# EPICS substitutions: plotApp/Db/plot.substitutions
# P comes from epicsEnvSet("P", ...) in st.cmd (e.g. TAS:Plot: or HB3:Plot:).
# Prefer one full prefix macro (HB3 Mot/Det/CS style), not Sys/Dev or P+R.
file "$(TOP)/plotApp/Db/plot.template"
{
pattern {P, MAXPTS, DATAFILETEXT}
{ $(P), 4000, 65536 }
}
